PROGRAM ModbusControl
VAR
	bWrite : BOOL;
	bRead: BOOL;
	fbMBwritereg : FB_MBWriteRegs;  
	fbMBreadreg : FB_MBReadRegs;
	adata : ARRAY [0..3] OF WORD;
	adatar : ARRAY [0..3] OF WORD;
	nQ : WORD :=4;
	estateread : StateMachineCommand;
	
	
END_VAR

GVL_Global.monitoringVAR.CurrentOpmod :=GVL_Global.commandsfromCLC.commands;
//GVL_Global.ModWrite.System_state_control  := GVL_Global.EthCommandsfrmCLC_IN.StatControlCMD;
GVL_Global.ModWrite.System_mode_control  := GVL_Global.EthCommandsfrmCLC_IN.OpModeControlCMD;
IF GVL_Global.bPower_enable = TRUE THEN
GVL_Global.ModWrite.Active_power_control := DINT_TO_INT(GVL_Global.EthCommandsfrmCLC_IN.ActivePowerReference)*10;
GVL_Global.ModWrite.Reactive_power_control := DINT_TO_INT(GVL_Global.EthCommandsfrmCLC_IN.ReactivePowerReference)*10;
ELSE
	GVL_Global.ModWrite.Active_power_control := 0;
GVL_Global.ModWrite.Reactive_power_control :=0;
END_IF
GVL_Global.ModWrite.Clear_fault := DINT_TO_USINT(GVL_Global.EthCommandsfrmCLC_IN.ClrFault);

IF NOT fbMBwritereg.bBusy THEN
	bWrite := TRUE;
fbMBwritereg(
	sIPAddr:= '10.200.8.219', //write at output reg of master i.e Eneraerk , CLC -- ws2lc
	nTCPPort:= 502, 
	nUnitID:= 255, 
	nQuantity:=SIZEOF(GVL_Global.ModWrite)/2, 
	nMBAddr:= 16#8020, 
	cbLength:= SIZEOF(GVL_Global.ModWrite), 
	pSrcAddr:= ADR(GVL_Global.ModWrite), 
	bExecute:= bWrite, 
	tTimeout:= T#5S, 
	bBusy=> , 
	bError=> , 
	nErrId=> );
	ELSE
		bWrite:= FALSE;
		fbMBwritereg(bExecute :=bWrite);
		
	END_IF
	
	IF NOT fbMBreadreg.bBusy THEN
		bRead := TRUE;
	fbMBreadreg(
	sIPAddr:= '10.200.8.219', 
	nTCPPort:= 502, 
	nUnitID:= 255, 
	nQuantity:= SIZEOF(GVL_Global.ModRead)/2, 
	nMBAddr:= 16#8000, 
	cbLength:= SIZEOF(GVL_Global.ModRead), 
	pDestAddr:= ADR(GVL_Global.ModRead), 
	bExecute:= bRead, 
	tTimeout:= T#5S, 
	bBusy=> , 
	bError=> , 
	nErrId=> , 
	cbRead=> );
	ELSE
		bRead := FALSE;
		fbMBreadreg(bExecute := bRead);
		
	END_IF
	//GVL_Higherlevel.enstate := WORD_TO_INT(adatar[0]);

END_PROGRAM

(* stored: Version 1.1.0.1, ProductVersion 3.1.4024.11
   POU ModbusControl: Id {5402e524-37ea-40bf-b0bd-a2aede11ed90}, SpecialFunc None *)
